KUKA KRL program: chk_w1_wechs_ok.src

&ACCESS RV12
&REL 5
&COMMENT Check C1
DEF chk_w1_wechs_ok( )
Diag_Appl(#on,5)

; VERIFICAÇÃO DE FERRAMENTA: C1

wait for (($in[161]) and (not $in[169]) and ($in[177]) and ($in[219]))

;//---- End -------
Diag_Appl(#Off,5)
END
